Omron CX-Programmer project NuevoProyecto (CX-Programmer 9.61)

# PLC NuevoPLC1: CQM1 CPU41

## Program NuevoPrograma1 (no task)
Local symbols
KMC 100.08 BOOL
KME 100.10 BOOL
KMI BOOL
KMT 100.09 BOOL
LAV 100.13 BOOL
LFUNC 100.14 BOOL
PM 0.08 BOOL
PP 0.15 BOOL
RT 0.13 BOOL

### Section Sección1

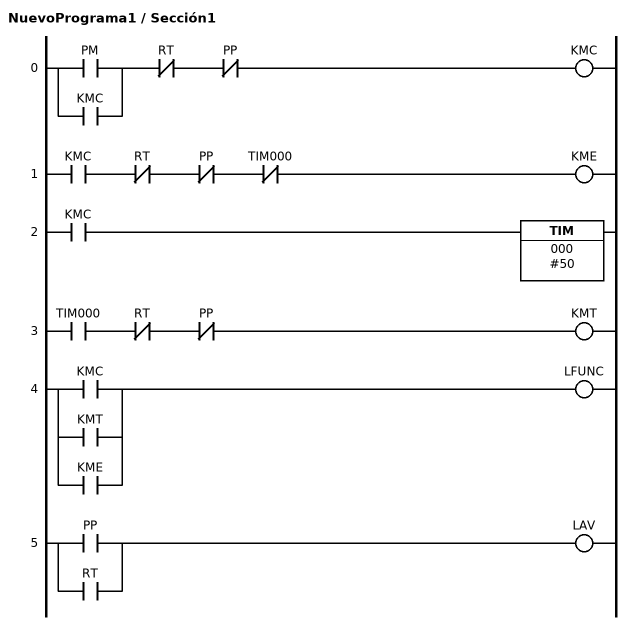
; rung 0
LD PM
OR KMC
ANDNOT RT
ANDNOT PP
OUT KMC
; rung 1
LD KMC
ANDNOT RT
ANDNOT PP
ANDNOT TIM000
OUT KME
; rung 2
LD KMC
TIM 000 #50
; rung 3
LD TIM000
ANDNOT RT
ANDNOT PP
OUT KMT
; rung 4
LD KMC
OR KMT
OR KME
OUT LFUNC
; rung 5
LD PP
OR RT
OUT LAV

### Section END
; rung 0
END(01)